(*
SPDX-FileCopyrightText: © 2026 Oleksandr Tiutyk <trofimich@gmail.com>
SPDX-License-Identifier: MIT
License: https://opensource.org/license/mit
*)

(*!
<summary>
Beckhoff EL4002_EX: Extended 2-channel analog output terminal with diagnostics.
</summary>
<description>
Extends EL4002 with EtherCAT Working Counter and slave state diagnostics.
When used for I/O, link located fields or their containing buffers to the matching selected PDOs.
The record is not a packed wire buffer; compiler padding is not part of the device specification.
Unlinked/default values do not prove valid I/O. The caller evaluates bus/channel validity before use.
Use one owner task per instance and externally synchronize other access; multi-field snapshots are not atomic.
Copies store data without creating hardware links. Keep borrowed field references valid while consumers are bound.
This passive record performs no validation, synchronization, configuration or protocol advancement.
WcState=TRUE means process-data exchange is invalid. State is acyclic EtherCAT/link information,
not proof of current measurement validity. Link diagnostics to the matching slave InfoData entries.
The selected PDO representation is documented by the base terminal model.
AdsAddr is acyclic mailbox addressing information, not a measurement-validity indicator.
Channels hold raw INT16 output commands; configure electrical range and presentation before use.
</description>
*)
TYPE EL4002_EX EXTENDS EL4002 :
STRUCT
	WcState AT %I* : BOOL;
	State AT %I* : UINT;
	AdsAddr AT %I* : Global.AMSADDR;
END_STRUCT
END_TYPE

(* stored: Version 1.1.0.1, ProductVersion 3.1.4026.18
   DUT EL4002_EX: Id {4ce337eb-dedb-4521-b806-1159fb1e34db} *)
